TYPE ST_EPSLimits :
STRUCT
	fFwd_Limits : REAL;
	fBwd_Limits	: REAL;
	fbEPS 		: FB_EPS;
END_STRUCT
END_TYPE

(* stored: Version 1.1.0.1, ProductVersion 3.1.4022.18
   DUT ST_EPSLimits: Id {4ee57205-73a9-412c-b8d8-c1dfce7e0790} *)
